// TIA Portal V20 export
FUNCTION "CallManualOperationLines_Unit1" : Void   // FC83, LAD
// stored: SetENOAutomatically false
   VAR_TEMP
      StatusEm : Array[0..7] of Struct
         Status : Array[0..40] of Word;
      END_STRUCT;
      errorIDEm : Array[0..7] of Struct
         errorID : Array[0..40] of Word;
      END_STRUCT;
      disableUnit1 : Bool;
      TempAxisCommands : "LBC_typeAxis64PosManualCommands";
      TempAxisMonitoring : "LBC_typeAxis64PosProcessValues";
      TempSoftCam : Array[0..8] of "LER_typeSoftCamParameter";
   END_VAR
   VAR CONSTANT
      MECHANIC_NAME_ENABLE : Bool;
   END_VAR
   VAR_TEMP   // added for the SCL form of the ladder/FBD networks
      _w1 : Bool;
   END_VAR
BEGIN

REGION Network 1: Unit 1 Enable Manual Operation
   // Condition to disable manual operation lines in Unit 3
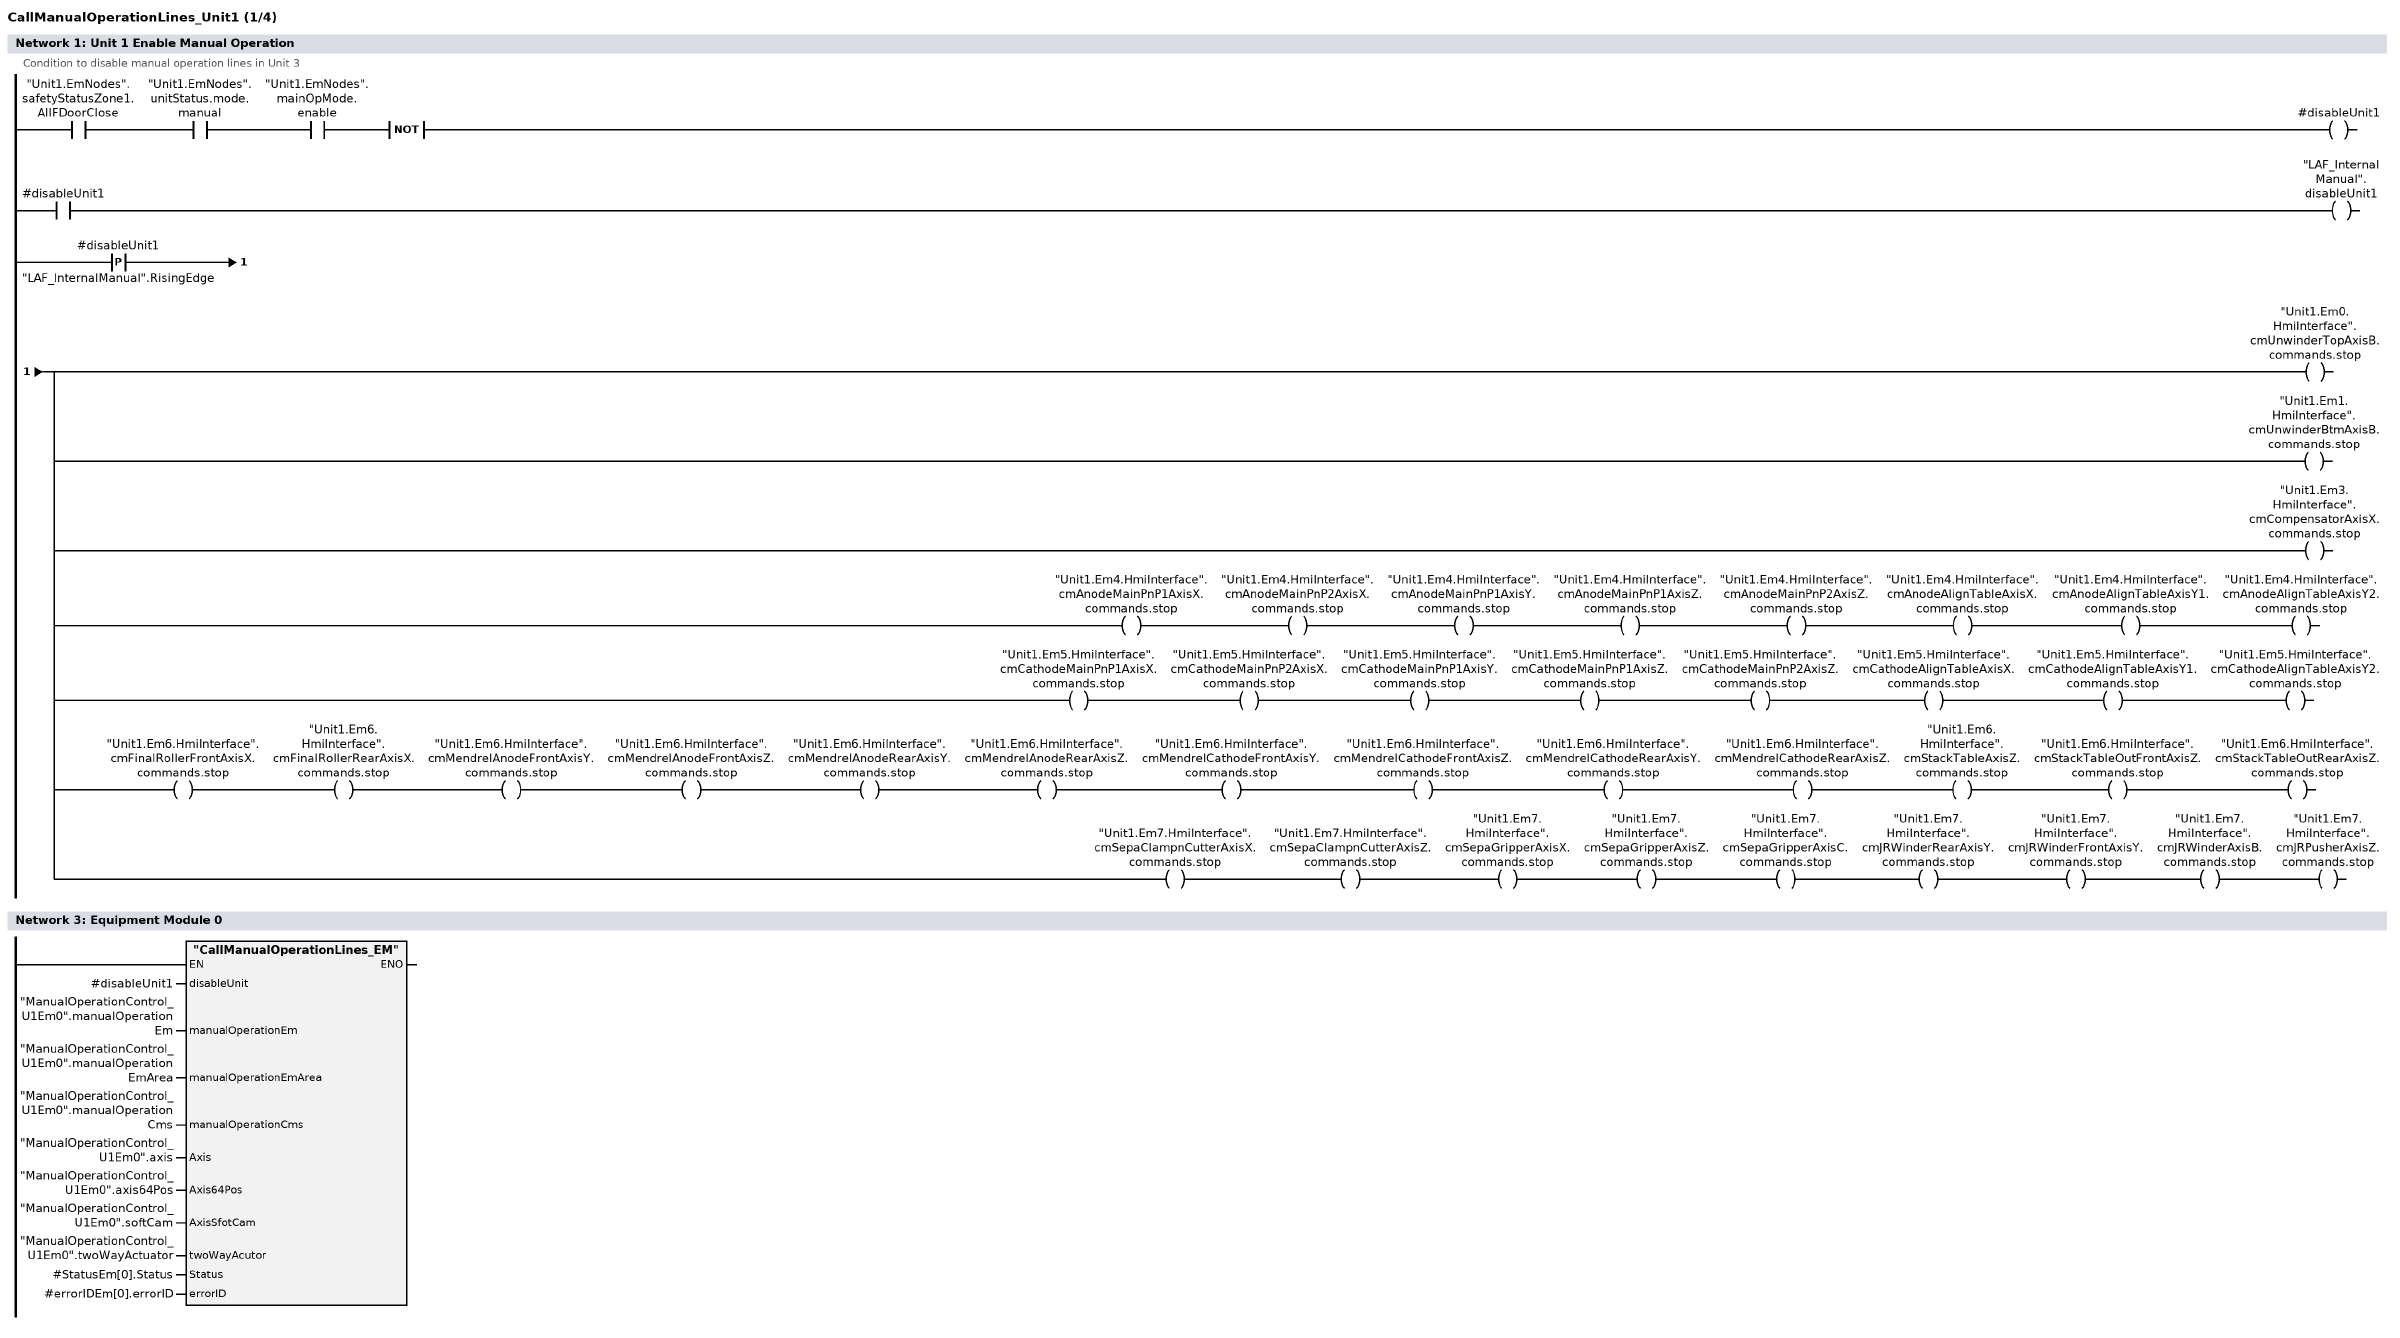
   RUNG wire#powerrail
      Contact( "Unit1.EmNodes".safetyStatusZone1.AllFDoorClose )
      Contact( "Unit1.EmNodes".unitStatus.mode.manual )
      Contact( "Unit1.EmNodes".mainOpMode.enable )
      Not()
      Coil( #disableUnit1 )
   END_RUNG
   RUNG wire#powerrail
      Contact( #disableUnit1 )
      Coil( "LAF_InternalManual".disableUnit1 )
   END_RUNG
   RUNG wire#powerrail
      P_Contact(operand := #disableUnit1, bit := "LAF_InternalManual".RisingEdge)
      wire#w1
      Coil( "Unit1.Em0.HmiInterface".cmUnwinderTopAxisB.commands.stop )
   END_RUNG
   RUNG wire#w1
      Coil( "Unit1.Em1.HmiInterface".cmUnwinderBtmAxisB.commands.stop )
   END_RUNG
   RUNG wire#w1
      Coil( "Unit1.Em3.HmiInterface".cmCompensatorAxisX.commands.stop )
   END_RUNG
   RUNG wire#w1
      Coil( "Unit1.Em4.HmiInterface".cmAnodeMainPnP1AxisX.commands.stop )
      Coil( "Unit1.Em4.HmiInterface".cmAnodeMainPnP2AxisX.commands.stop )
      Coil( "Unit1.Em4.HmiInterface".cmAnodeMainPnP1AxisY.commands.stop )
      Coil( "Unit1.Em4.HmiInterface".cmAnodeMainPnP1AxisZ.commands.stop )
      Coil( "Unit1.Em4.HmiInterface".cmAnodeMainPnP2AxisZ.commands.stop )
      Coil( "Unit1.Em4.HmiInterface".cmAnodeAlignTableAxisX.commands.stop )
      Coil( "Unit1.Em4.HmiInterface".cmAnodeAlignTableAxisY1.commands.stop )
      Coil( "Unit1.Em4.HmiInterface".cmAnodeAlignTableAxisY2.commands.stop )
   END_RUNG
   RUNG wire#w1
      Coil( "Unit1.Em5.HmiInterface".cmCathodeMainPnP1AxisX.commands.stop )
      Coil( "Unit1.Em5.HmiInterface".cmCathodeMainPnP2AxisX.commands.stop )
      Coil( "Unit1.Em5.HmiInterface".cmCathodeMainPnP1AxisY.commands.stop )
      Coil( "Unit1.Em5.HmiInterface".cmCathodeMainPnP1AxisZ.commands.stop )
      Coil( "Unit1.Em5.HmiInterface".cmCathodeMainPnP2AxisZ.commands.stop )
      Coil( "Unit1.Em5.HmiInterface".cmCathodeAlignTableAxisX.commands.stop )
      Coil( "Unit1.Em5.HmiInterface".cmCathodeAlignTableAxisY1.commands.stop )
      Coil( "Unit1.Em5.HmiInterface".cmCathodeAlignTableAxisY2.commands.stop )
   END_RUNG
   RUNG wire#w1
      Coil( "Unit1.Em6.HmiInterface".cmFinalRollerFrontAxisX.commands.stop )
      Coil( "Unit1.Em6.HmiInterface".cmFinalRollerRearAxisX.commands.stop )
      Coil( "Unit1.Em6.HmiInterface".cmMendrelAnodeFrontAxisY.commands.stop )
      Coil( "Unit1.Em6.HmiInterface".cmMendrelAnodeFrontAxisZ.commands.stop )
      Coil( "Unit1.Em6.HmiInterface".cmMendrelAnodeRearAxisY.commands.stop )
      Coil( "Unit1.Em6.HmiInterface".cmMendrelAnodeRearAxisZ.commands.stop )
      Coil( "Unit1.Em6.HmiInterface".cmMendrelCathodeFrontAxisY.commands.stop )
      Coil( "Unit1.Em6.HmiInterface".cmMendrelCathodeFrontAxisZ.commands.stop )
      Coil( "Unit1.Em6.HmiInterface".cmMendrelCathodeRearAxisY.commands.stop )
      Coil( "Unit1.Em6.HmiInterface".cmMendrelCathodeRearAxisZ.commands.stop )
      Coil( "Unit1.Em6.HmiInterface".cmStackTableAxisZ.commands.stop )
      Coil( "Unit1.Em6.HmiInterface".cmStackTableOutFrontAxisZ.commands.stop )
      Coil( "Unit1.Em6.HmiInterface".cmStackTableOutRearAxisZ.commands.stop )
   END_RUNG
   RUNG wire#w1
      Coil( "Unit1.Em7.HmiInterface".cmSepaClampnCutterAxisX.commands.stop )
      Coil( "Unit1.Em7.HmiInterface".cmSepaClampnCutterAxisZ.commands.stop )
      Coil( "Unit1.Em7.HmiInterface".cmSepaGripperAxisX.commands.stop )
      Coil( "Unit1.Em7.HmiInterface".cmSepaGripperAxisZ.commands.stop )
      Coil( "Unit1.Em7.HmiInterface".cmSepaGripperAxisC.commands.stop )
      Coil( "Unit1.Em7.HmiInterface".cmJRWinderRearAxisY.commands.stop )
      Coil( "Unit1.Em7.HmiInterface".cmJRWinderFrontAxisY.commands.stop )
      Coil( "Unit1.Em7.HmiInterface".cmJRWinderAxisB.commands.stop )
      Coil( "Unit1.Em7.HmiInterface".cmJRPusherAxisZ.commands.stop )
   END_RUNG
   // the same network as SCL:
   #disableUnit1 := NOT ("Unit1.EmNodes".safetyStatusZone1.AllFDoorClose AND "Unit1.EmNodes".unitStatus.mode.manual AND "Unit1.EmNodes".mainOpMode.enable);
   "LAF_InternalManual".disableUnit1 := #disableUnit1;
   #_w1 := #disableUnit1 AND NOT "LAF_InternalManual".RisingEdge;   // rising edge of #disableUnit1
   "LAF_InternalManual".RisingEdge := #disableUnit1;
   "Unit1.Em0.HmiInterface".cmUnwinderTopAxisB.commands.stop := #_w1;
   "Unit1.Em1.HmiInterface".cmUnwinderBtmAxisB.commands.stop := #_w1;
   "Unit1.Em3.HmiInterface".cmCompensatorAxisX.commands.stop := #_w1;
   "Unit1.Em4.HmiInterface".cmAnodeMainPnP1AxisX.commands.stop := #_w1;
   "Unit1.Em4.HmiInterface".cmAnodeMainPnP2AxisX.commands.stop := #_w1;
   "Unit1.Em4.HmiInterface".cmAnodeMainPnP1AxisY.commands.stop := #_w1;
   "Unit1.Em4.HmiInterface".cmAnodeMainPnP1AxisZ.commands.stop := #_w1;
   "Unit1.Em4.HmiInterface".cmAnodeMainPnP2AxisZ.commands.stop := #_w1;
   "Unit1.Em4.HmiInterface".cmAnodeAlignTableAxisX.commands.stop := #_w1;
   "Unit1.Em4.HmiInterface".cmAnodeAlignTableAxisY1.commands.stop := #_w1;
   "Unit1.Em4.HmiInterface".cmAnodeAlignTableAxisY2.commands.stop := #_w1;
   "Unit1.Em5.HmiInterface".cmCathodeMainPnP1AxisX.commands.stop := #_w1;
   "Unit1.Em5.HmiInterface".cmCathodeMainPnP2AxisX.commands.stop := #_w1;
   "Unit1.Em5.HmiInterface".cmCathodeMainPnP1AxisY.commands.stop := #_w1;
   "Unit1.Em5.HmiInterface".cmCathodeMainPnP1AxisZ.commands.stop := #_w1;
   "Unit1.Em5.HmiInterface".cmCathodeMainPnP2AxisZ.commands.stop := #_w1;
   "Unit1.Em5.HmiInterface".cmCathodeAlignTableAxisX.commands.stop := #_w1;
   "Unit1.Em5.HmiInterface".cmCathodeAlignTableAxisY1.commands.stop := #_w1;
   "Unit1.Em5.HmiInterface".cmCathodeAlignTableAxisY2.commands.stop := #_w1;
   "Unit1.Em6.HmiInterface".cmFinalRollerFrontAxisX.commands.stop := #_w1;
   "Unit1.Em6.HmiInterface".cmFinalRollerRearAxisX.commands.stop := #_w1;
   "Unit1.Em6.HmiInterface".cmMendrelAnodeFrontAxisY.commands.stop := #_w1;
   "Unit1.Em6.HmiInterface".cmMendrelAnodeFrontAxisZ.commands.stop := #_w1;
   "Unit1.Em6.HmiInterface".cmMendrelAnodeRearAxisY.commands.stop := #_w1;
   "Unit1.Em6.HmiInterface".cmMendrelAnodeRearAxisZ.commands.stop := #_w1;
   "Unit1.Em6.HmiInterface".cmMendrelCathodeFrontAxisY.commands.stop := #_w1;
   "Unit1.Em6.HmiInterface".cmMendrelCathodeFrontAxisZ.commands.stop := #_w1;
   "Unit1.Em6.HmiInterface".cmMendrelCathodeRearAxisY.commands.stop := #_w1;
   "Unit1.Em6.HmiInterface".cmMendrelCathodeRearAxisZ.commands.stop := #_w1;
   "Unit1.Em6.HmiInterface".cmStackTableAxisZ.commands.stop := #_w1;
   "Unit1.Em6.HmiInterface".cmStackTableOutFrontAxisZ.commands.stop := #_w1;
   "Unit1.Em6.HmiInterface".cmStackTableOutRearAxisZ.commands.stop := #_w1;
   "Unit1.Em7.HmiInterface".cmSepaClampnCutterAxisX.commands.stop := #_w1;
   "Unit1.Em7.HmiInterface".cmSepaClampnCutterAxisZ.commands.stop := #_w1;
   "Unit1.Em7.HmiInterface".cmSepaGripperAxisX.commands.stop := #_w1;
   "Unit1.Em7.HmiInterface".cmSepaGripperAxisZ.commands.stop := #_w1;
   "Unit1.Em7.HmiInterface".cmSepaGripperAxisC.commands.stop := #_w1;
   "Unit1.Em7.HmiInterface".cmJRWinderRearAxisY.commands.stop := #_w1;
   "Unit1.Em7.HmiInterface".cmJRWinderFrontAxisY.commands.stop := #_w1;
   "Unit1.Em7.HmiInterface".cmJRWinderAxisB.commands.stop := #_w1;
   "Unit1.Em7.HmiInterface".cmJRPusherAxisZ.commands.stop := #_w1;
END_REGION

REGION Network 2 (SCL): Equipment Module 0 Cms Mapping
   REGION Input Mapping
       // Axis
       "ManualOperationControl_U1Em0".axis64Pos[6].monitoring := "Unit1.Em0.HmiInterface".cmUnwinderTopAxisB.monitoring;

       "ManualOperationControl_U1Em0".axis64Pos[6].configuration := "Unit1.Em0.HmiInterface".cmUnwinderTopAxisB.configuration;
       // SoftCam
       "ManualOperationControl_U1Em0".softCam[6] := "Unit1.Em0.HmiInterface".cm.softCam.unwinderTopAxisB;

       // TwoWayActuator
       "ManualOperationControl_U1Em0".twoWayActuator[1].monitoring := "Unit1.Em0.HmiInterface".cmAirShaftTopOnOff.monitoring;
   END_REGION


   REGION Output Mapping
       // Axis
       "CallManualOperationLines_ServoPos64Commands"(ManualOperationControl := "ManualOperationControl_U1Em0".axis64Pos[6].commands,
                                                     HmiInterface => "Unit1.Em0.HmiInterface".cmUnwinderTopAxisB.commands);

       // TwoWayActuator
       "Unit1.Em0.HmiInterface".cmAirShaftTopOnOff.commands := "ManualOperationControl_U1Em0".twoWayActuator[1].commands;
   END_REGION
END_REGION

REGION Network 3: Equipment Module 0
   RUNG wire#powerrail
      "CallManualOperationLines_EM"(disableUnit := #disableUnit1, manualOperationEm := "ManualOperationControl_U1Em0".manualOperationEm, manualOperationEmArea := "ManualOperationControl_U1Em0".manualOperationEmArea, manualOperationCms := "ManualOperationControl_U1Em0".manualOperationCms, Axis := "ManualOperationControl_U1Em0".axis, Axis64Pos := "ManualOperationControl_U1Em0".axis64Pos, AxisSfotCam := "ManualOperationControl_U1Em0".softCam, twoWayAcutor := "ManualOperationControl_U1Em0".twoWayActuator, Status := #StatusEm[0].Status, errorID := #errorIDEm[0].errorID)
   END_RUNG
   // the same network as SCL:
   "CallManualOperationLines_EM"(disableUnit := #disableUnit1,
                           manualOperationEm := "ManualOperationControl_U1Em0".manualOperationEm,
                           manualOperationEmArea := "ManualOperationControl_U1Em0".manualOperationEmArea,
                           manualOperationCms := "ManualOperationControl_U1Em0".manualOperationCms,
                           Axis := "ManualOperationControl_U1Em0".axis,
                           Axis64Pos := "ManualOperationControl_U1Em0".axis64Pos,
                           AxisSfotCam := "ManualOperationControl_U1Em0".softCam,
                           twoWayAcutor := "ManualOperationControl_U1Em0".twoWayActuator,
                           Status := #StatusEm[0].Status,
                           errorID := #errorIDEm[0].errorID);
END_REGION

REGION Network 4 (SCL): Equipment Module 1 Cms Mapping
   REGION Input Mapping
       // Axis
       "ManualOperationControl_U1Em1".axis64Pos[6].monitoring := "Unit1.Em1.HmiInterface".cmUnwinderBtmAxisB.monitoring;

       "ManualOperationControl_U1Em1".axis64Pos[6].configuration := "Unit1.Em1.HmiInterface".cmUnwinderBtmAxisB.configuration;
       // SoftCam
       "ManualOperationControl_U1Em1".softCam[6] := "Unit1.Em1.HmiInterface".cm.softCam.unwinderBtmAxisB;

       // TwoWayActuator
       "ManualOperationControl_U1Em1".twoWayActuator[1].monitoring := "Unit1.Em1.HmiInterface".cmAirShaftBtmOnOff.monitoring;
   END_REGION


   REGION Output Mapping
       // Axis
       "CallManualOperationLines_ServoPos64Commands"(ManualOperationControl := "ManualOperationControl_U1Em1".axis64Pos[6].commands,
                                                     HmiInterface => "Unit1.Em1.HmiInterface".cmUnwinderBtmAxisB.commands);

       // TwoWayActuator
       "Unit1.Em0.HmiInterface".cmAirShaftTopOnOff.commands := "ManualOperationControl_U1Em0".twoWayActuator[1].commands;
   END_REGION
END_REGION

REGION Network 5: Equipment Module 1
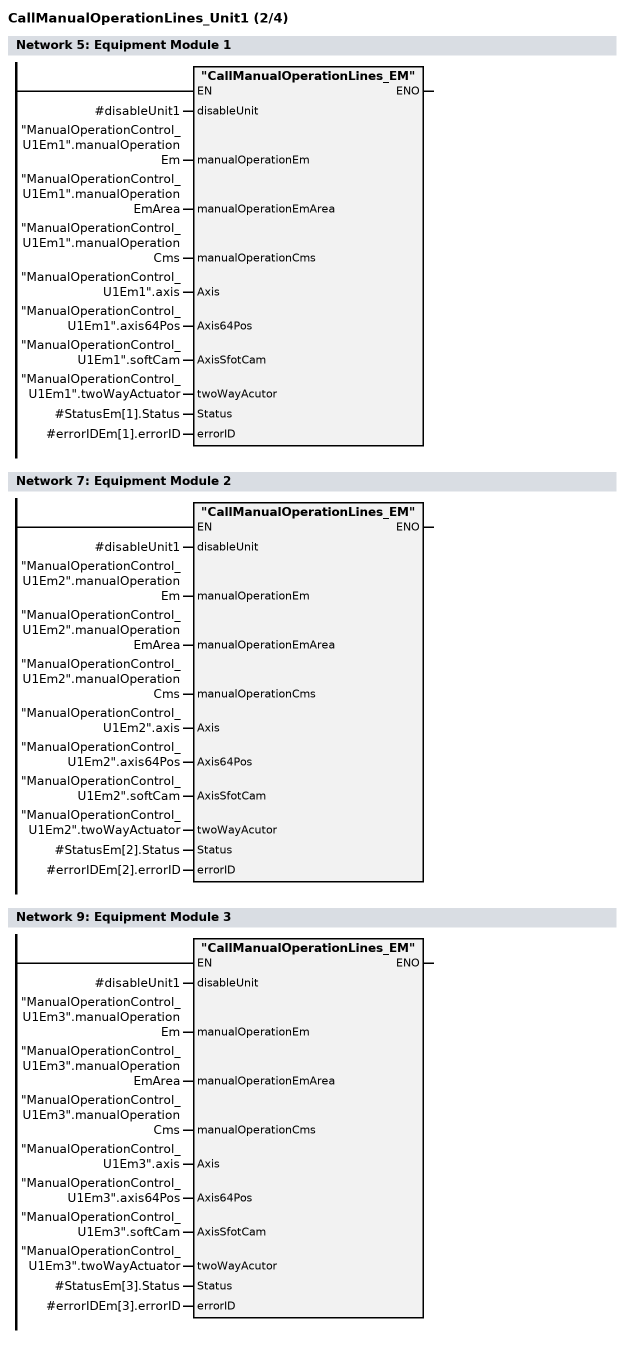
   RUNG wire#powerrail
      "CallManualOperationLines_EM"(disableUnit := #disableUnit1, manualOperationEm := "ManualOperationControl_U1Em1".manualOperationEm, manualOperationEmArea := "ManualOperationControl_U1Em1".manualOperationEmArea, manualOperationCms := "ManualOperationControl_U1Em1".manualOperationCms, Axis := "ManualOperationControl_U1Em1".axis, Axis64Pos := "ManualOperationControl_U1Em1".axis64Pos, AxisSfotCam := "ManualOperationControl_U1Em1".softCam, twoWayAcutor := "ManualOperationControl_U1Em1".twoWayActuator, Status := #StatusEm[1].Status, errorID := #errorIDEm[1].errorID)
   END_RUNG
   // the same network as SCL:
   "CallManualOperationLines_EM"(disableUnit := #disableUnit1,
                           manualOperationEm := "ManualOperationControl_U1Em1".manualOperationEm,
                           manualOperationEmArea := "ManualOperationControl_U1Em1".manualOperationEmArea,
                           manualOperationCms := "ManualOperationControl_U1Em1".manualOperationCms,
                           Axis := "ManualOperationControl_U1Em1".axis,
                           Axis64Pos := "ManualOperationControl_U1Em1".axis64Pos,
                           AxisSfotCam := "ManualOperationControl_U1Em1".softCam,
                           twoWayAcutor := "ManualOperationControl_U1Em1".twoWayActuator,
                           Status := #StatusEm[1].Status,
                           errorID := #errorIDEm[1].errorID);
END_REGION

REGION Network 6 (SCL): Equipment Module 2 Cms Mapping
   REGION Input Mapping  
       // TwoWayActuator
       "ManualOperationControl_U1Em2".twoWayActuator[1].monitoring := "Unit1.Em2.HmiInterface".cmSuctionPadTopUpDown.monitoring;
       "ManualOperationControl_U1Em2".twoWayActuator[2].monitoring := "Unit1.Em2.HmiInterface".cmSuctionPadBtmUpDown.monitoring;
       "ManualOperationControl_U1Em2".twoWayActuator[3].monitoring := "Unit1.Em2.HmiInterface".cmCutterUpDown.monitoring;
       "ManualOperationControl_U1Em2".twoWayActuator[4].monitoring := "Unit1.Em2.HmiInterface".cmTapeTopUpDown.monitoring;
       "ManualOperationControl_U1Em2".twoWayActuator[5].monitoring := "Unit1.Em2.HmiInterface".cmTapeBtmUpDown.monitoring;
       "ManualOperationControl_U1Em2".twoWayActuator[6].monitoring := "Unit1.Em2.HmiInterface".cmSpliceHeadRotateTopFwdBwd.monitoring;
       "ManualOperationControl_U1Em2".twoWayActuator[7].monitoring := "Unit1.Em2.HmiInterface".cmSpliceHeadRotateBtmFwdBwd.monitoring;
       "ManualOperationControl_U1Em2".twoWayActuator[8].monitoring := "Unit1.Em2.HmiInterface".cmSuctionPadTopLeftVaccum.monitoring;
       "ManualOperationControl_U1Em2".twoWayActuator[9].monitoring := "Unit1.Em2.HmiInterface".cmSuctionPadTopRightVaccum.monitoring;
       "ManualOperationControl_U1Em2".twoWayActuator[10].monitoring := "Unit1.Em2.HmiInterface".cmSuctionPadBtmLeftVaccum.monitoring;
       "ManualOperationControl_U1Em2".twoWayActuator[11].monitoring := "Unit1.Em2.HmiInterface".cmSuctionPadBtmRightVaccum.monitoring;
       "ManualOperationControl_U1Em2".twoWayActuator[12].monitoring := "Unit1.Em2.HmiInterface".cmSuctionPadTopTapeVaccum.monitoring;
       "ManualOperationControl_U1Em2".twoWayActuator[13].monitoring := "Unit1.Em2.HmiInterface".cmSuctionPadBtmTapeVaccum.monitoring;

   END_REGION

   REGION Output Mapping
       // TwoWayActuator
       "Unit1.Em2.HmiInterface".cmSuctionPadTopUpDown.commands := "ManualOperationControl_U1Em2".twoWayActuator[1].commands;
       "Unit1.Em2.HmiInterface".cmSuctionPadBtmUpDown.commands := "ManualOperationControl_U1Em2".twoWayActuator[2].commands;
       "Unit1.Em2.HmiInterface".cmCutterUpDown.commands := "ManualOperationControl_U1Em2".twoWayActuator[3].commands;
       "Unit1.Em2.HmiInterface".cmTapeTopUpDown.commands := "ManualOperationControl_U1Em2".twoWayActuator[4].commands;
       "Unit1.Em2.HmiInterface".cmTapeBtmUpDown.commands := "ManualOperationControl_U1Em2".twoWayActuator[5].commands;
       "Unit1.Em2.HmiInterface".cmSpliceHeadRotateTopFwdBwd.commands := "ManualOperationControl_U1Em2".twoWayActuator[6].commands;
       "Unit1.Em2.HmiInterface".cmSpliceHeadRotateBtmFwdBwd.commands := "ManualOperationControl_U1Em2".twoWayActuator[7].commands;
       "Unit1.Em2.HmiInterface".cmSuctionPadTopLeftVaccum.commands := "ManualOperationControl_U1Em2".twoWayActuator[8].commands;
       "Unit1.Em2.HmiInterface".cmSuctionPadTopRightVaccum.commands := "ManualOperationControl_U1Em2".twoWayActuator[9].commands;
       "Unit1.Em2.HmiInterface".cmSuctionPadBtmLeftVaccum.commands := "ManualOperationControl_U1Em2".twoWayActuator[10].commands;
       "Unit1.Em2.HmiInterface".cmSuctionPadBtmRightVaccum.commands := "ManualOperationControl_U1Em2".twoWayActuator[11].commands;
       "Unit1.Em2.HmiInterface".cmSuctionPadTopTapeVaccum.commands := "ManualOperationControl_U1Em2".twoWayActuator[12].commands;
       "Unit1.Em2.HmiInterface".cmSuctionPadBtmTapeVaccum.commands := "ManualOperationControl_U1Em2".twoWayActuator[13].commands;

   END_REGION
END_REGION

REGION Network 7: Equipment Module 2
   RUNG wire#powerrail
      "CallManualOperationLines_EM"(disableUnit := #disableUnit1, manualOperationEm := "ManualOperationControl_U1Em2".manualOperationEm, manualOperationEmArea := "ManualOperationControl_U1Em2".manualOperationEmArea, manualOperationCms := "ManualOperationControl_U1Em2".manualOperationCms, Axis := "ManualOperationControl_U1Em2".axis, Axis64Pos := "ManualOperationControl_U1Em2".axis64Pos, AxisSfotCam := "ManualOperationControl_U1Em2".softCam, twoWayAcutor := "ManualOperationControl_U1Em2".twoWayActuator, Status := #StatusEm[2].Status, errorID := #errorIDEm[2].errorID)
   END_RUNG
   // the same network as SCL:
   "CallManualOperationLines_EM"(disableUnit := #disableUnit1,
                           manualOperationEm := "ManualOperationControl_U1Em2".manualOperationEm,
                           manualOperationEmArea := "ManualOperationControl_U1Em2".manualOperationEmArea,
                           manualOperationCms := "ManualOperationControl_U1Em2".manualOperationCms,
                           Axis := "ManualOperationControl_U1Em2".axis,
                           Axis64Pos := "ManualOperationControl_U1Em2".axis64Pos,
                           AxisSfotCam := "ManualOperationControl_U1Em2".softCam,
                           twoWayAcutor := "ManualOperationControl_U1Em2".twoWayActuator,
                           Status := #StatusEm[2].Status,
                           errorID := #errorIDEm[2].errorID);
END_REGION

REGION Network 8 (SCL): Equipment Module 3 Cms Mapping
   REGION Input Mapping
       // Axis
       "ManualOperationControl_U1Em3".axis64Pos[6].monitoring := "Unit1.Em3.HmiInterface".cmCompensatorAxisX.monitoring;
       //"ManualOperationControl_U1Em3".axis[2].monitoring := Unit1.Em3.HmiInterface.cmSepaFeedingRollerAxisB.monitoring;
       "ManualOperationControl_U1Em3".axis64Pos[6].configuration := "Unit1.Em3.HmiInterface".cmCompensatorAxisX.configuration;
       // SoftCam
       "ManualOperationControl_U1Em3".softCam[6] := "Unit1.Em3.HmiInterface".cm.softCam.compensatorAxisX;

       // TwoWayActuator
       "ManualOperationControl_U1Em3".twoWayActuator[1].monitoring := "Unit1.Em3.HmiInterface".cmDancerFwdBwd.monitoring;
       "ManualOperationControl_U1Em3".twoWayActuator[2].monitoring := "Unit1.Em3.HmiInterface".cmSepaUnwinderIonizerTop.monitoring;
       "ManualOperationControl_U1Em3".twoWayActuator[3].monitoring := "Unit1.Em3.HmiInterface".cmSepaUnwinderIonizerBottom.monitoring;

   END_REGION

   REGION Output Mapping
       // Axis
       "CallManualOperationLines_ServoPos64Commands"(ManualOperationControl := "ManualOperationControl_U1Em3".axis64Pos[6].commands,
                                                     HmiInterface => "Unit1.Em3.HmiInterface".cmCompensatorAxisX.commands);

       // TwoWayActuator
       "Unit1.Em3.HmiInterface".cmDancerFwdBwd.commands := "ManualOperationControl_U1Em3".twoWayActuator[1].commands;
       "Unit1.Em3.HmiInterface".cmSepaUnwinderIonizerTop.commands := "ManualOperationControl_U1Em3".twoWayActuator[2].commands;
       "Unit1.Em3.HmiInterface".cmSepaUnwinderIonizerBottom.commands := "ManualOperationControl_U1Em3".twoWayActuator[3].commands;

   END_REGION
END_REGION

REGION Network 9: Equipment Module 3
   RUNG wire#powerrail
      "CallManualOperationLines_EM"(disableUnit := #disableUnit1, manualOperationEm := "ManualOperationControl_U1Em3".manualOperationEm, manualOperationEmArea := "ManualOperationControl_U1Em3".manualOperationEmArea, manualOperationCms := "ManualOperationControl_U1Em3".manualOperationCms, Axis := "ManualOperationControl_U1Em3".axis, Axis64Pos := "ManualOperationControl_U1Em3".axis64Pos, AxisSfotCam := "ManualOperationControl_U1Em3".softCam, twoWayAcutor := "ManualOperationControl_U1Em3".twoWayActuator, Status := #StatusEm[3].Status, errorID := #errorIDEm[3].errorID)
   END_RUNG
   // the same network as SCL:
   "CallManualOperationLines_EM"(disableUnit := #disableUnit1,
                           manualOperationEm := "ManualOperationControl_U1Em3".manualOperationEm,
                           manualOperationEmArea := "ManualOperationControl_U1Em3".manualOperationEmArea,
                           manualOperationCms := "ManualOperationControl_U1Em3".manualOperationCms,
                           Axis := "ManualOperationControl_U1Em3".axis,
                           Axis64Pos := "ManualOperationControl_U1Em3".axis64Pos,
                           AxisSfotCam := "ManualOperationControl_U1Em3".softCam,
                           twoWayAcutor := "ManualOperationControl_U1Em3".twoWayActuator,
                           Status := #StatusEm[3].Status,
                           errorID := #errorIDEm[3].errorID);
END_REGION

REGION Network 10 (SCL): Equipment Module 4 Cms Mapping
   REGION Input Mapping
       // Axis
       "ManualOperationControl_U1Em4".axis64Pos[6].monitoring := "Unit1.Em4.HmiInterface".cmAnodeMainPnP1AxisX.monitoring;
       "ManualOperationControl_U1Em4".axis64Pos[7].monitoring := "Unit1.Em4.HmiInterface".cmAnodeMainPnP2AxisX.monitoring;
       "ManualOperationControl_U1Em4".axis64Pos[8].monitoring := "Unit1.Em4.HmiInterface".cmAnodeMainPnP1AxisY.monitoring;
       "ManualOperationControl_U1Em4".axis64Pos[9].monitoring := "Unit1.Em4.HmiInterface".cmAnodeMainPnP1AxisZ.monitoring;
       "ManualOperationControl_U1Em4".axis64Pos[10].monitoring := "Unit1.Em4.HmiInterface".cmAnodeMainPnP2AxisZ.monitoring;
       "ManualOperationControl_U1Em4".axis64Pos[11].monitoring := "Unit1.Em4.HmiInterface".cmAnodeAlignTableAxisX.monitoring;
       "ManualOperationControl_U1Em4".axis64Pos[12].monitoring := "Unit1.Em4.HmiInterface".cmAnodeAlignTableAxisY1.monitoring;
       "ManualOperationControl_U1Em4".axis64Pos[13].monitoring := "Unit1.Em4.HmiInterface".cmAnodeAlignTableAxisY2.monitoring;

       "ManualOperationControl_U1Em4".axis64Pos[6].configuration := "Unit1.Em4.HmiInterface".cmAnodeMainPnP1AxisX.configuration;
       "ManualOperationControl_U1Em4".axis64Pos[7].configuration := "Unit1.Em4.HmiInterface".cmAnodeMainPnP2AxisX.configuration;
       "ManualOperationControl_U1Em4".axis64Pos[8].configuration := "Unit1.Em4.HmiInterface".cmAnodeMainPnP1AxisY.configuration;
       "ManualOperationControl_U1Em4".axis64Pos[9].configuration := "Unit1.Em4.HmiInterface".cmAnodeMainPnP1AxisZ.configuration;
       "ManualOperationControl_U1Em4".axis64Pos[10].configuration := "Unit1.Em4.HmiInterface".cmAnodeMainPnP2AxisZ.configuration;
       "ManualOperationControl_U1Em4".axis64Pos[11].configuration := "Unit1.Em4.HmiInterface".cmAnodeAlignTableAxisX.configuration;
       "ManualOperationControl_U1Em4".axis64Pos[12].configuration := "Unit1.Em4.HmiInterface".cmAnodeAlignTableAxisY1.configuration;
       "ManualOperationControl_U1Em4".axis64Pos[13].configuration := "Unit1.Em4.HmiInterface".cmAnodeAlignTableAxisY2.configuration;

       // SoftCam
       "ManualOperationControl_U1Em4".softCam[6] := "Unit1.Em4.HmiInterface".cm.softCam.anodeMainPnP1AxisX;
       "ManualOperationControl_U1Em4".softCam[7] := "Unit1.Em4.HmiInterface".cm.softCam.anodeMainPnP2AxisX;
       "ManualOperationControl_U1Em4".softCam[8] := "Unit1.Em4.HmiInterface".cm.softCam.anodeMainPnP1AxisY;
       "ManualOperationControl_U1Em4".softCam[9] := "Unit1.Em4.HmiInterface".cm.softCam.anodeMainPnP1AxisZ;
       "ManualOperationControl_U1Em4".softCam[10] := "Unit1.Em4.HmiInterface".cm.softCam.anodeMainPnP2AxisZ;
       "ManualOperationControl_U1Em4".softCam[11] := "Unit1.Em4.HmiInterface".cm.softCam.anodeAlignTableAxisX;
       "ManualOperationControl_U1Em4".softCam[12] := "Unit1.Em4.HmiInterface".cm.softCam.anodeAlignTableAxisY1;
       "ManualOperationControl_U1Em4".softCam[13] := "Unit1.Em4.HmiInterface".cm.softCam.anodeAlignTableAxisY2;

       // TwoWayActuator
       "ManualOperationControl_U1Em4".twoWayActuator[1].monitoring := "Unit1.Em4.HmiInterface".cmAnodeMainPnP1RotaryCwCcw.monitoring;
       "ManualOperationControl_U1Em4".twoWayActuator[2].monitoring := "Unit1.Em4.HmiInterface".cmAnodeMainPnP1SuctionPlateVacuum.monitoring;
       "ManualOperationControl_U1Em4".twoWayActuator[3].monitoring := "Unit1.Em4.HmiInterface".cmAnodeMainPnP2SuctionPlateVacuum.monitoring;
       "ManualOperationControl_U1Em4".twoWayActuator[4].monitoring := "Unit1.Em4.HmiInterface".cmAnodeAlignTableSuctionPlateVacuum.monitoring;
       "ManualOperationControl_U1Em4".twoWayActuator[5].monitoring := "Unit1.Em4.HmiInterface".cmAnodeGlassCleaning.monitoring;
       "ManualOperationControl_U1Em4".twoWayActuator[6].monitoring := "Unit1.Em4.HmiInterface".cmAnodeNgPnpUpDown.monitoring;
       "ManualOperationControl_U1Em4".twoWayActuator[7].monitoring := "Unit1.Em4.HmiInterface".cmAnodeNgPnp1stFwdBwd.monitoring;
       "ManualOperationControl_U1Em4".twoWayActuator[8].monitoring := "Unit1.Em4.HmiInterface".cmAnodeNgPnp2ndFwdBwd.monitoring;
       "ManualOperationControl_U1Em4".twoWayActuator[9].monitoring := "Unit1.Em4.HmiInterface".cmAnodeMaintenanceMovingFixFrontRearFwdBwd.monitoring;
       "ManualOperationControl_U1Em4".twoWayActuator[10].monitoring := "Unit1.Em4.HmiInterface".cmAnodeNgBoxLiftUpDown.monitoring;
       "ManualOperationControl_U1Em4".twoWayActuator[11].monitoring := "Unit1.Em4.HmiInterface".cmAnodeNgBoxLockUpDown.monitoring;
       "ManualOperationControl_U1Em4".twoWayActuator[12].monitoring := "Unit1.Em4.HmiInterface".cmAnodeNgPnpVaccum.monitoring;
       "ManualOperationControl_U1Em4".twoWayActuator[13].monitoring := "Unit1.Em4.HmiInterface".cmAnodeConveyorCoverFwdBwd.monitoring;

   END_REGION


   REGION Output Mapping
       // Axis

       "CallManualOperationLines_ServoPos64Commands"(ManualOperationControl := "ManualOperationControl_U1Em4".axis64Pos[6].commands,
                                                     HmiInterface => "Unit1.Em4.HmiInterface".cmAnodeMainPnP1AxisX.commands);

       "CallManualOperationLines_ServoPos64Commands"(ManualOperationControl := "ManualOperationControl_U1Em4".axis64Pos[7].commands,
                                                     HmiInterface => "Unit1.Em4.HmiInterface".cmAnodeMainPnP2AxisX.commands);

       "CallManualOperationLines_ServoPos64Commands"(ManualOperationControl := "ManualOperationControl_U1Em4".axis64Pos[8].commands,
                                                     HmiInterface => "Unit1.Em4.HmiInterface".cmAnodeMainPnP1AxisY.commands);

       "CallManualOperationLines_ServoPos64Commands"(ManualOperationControl := "ManualOperationControl_U1Em4".axis64Pos[9].commands,
                                                     HmiInterface => "Unit1.Em4.HmiInterface".cmAnodeMainPnP1AxisZ.commands);

       "CallManualOperationLines_ServoPos64Commands"(ManualOperationControl := "ManualOperationControl_U1Em4".axis64Pos[10].commands,
                                                     HmiInterface => "Unit1.Em4.HmiInterface".cmAnodeMainPnP2AxisZ.commands);

       "CallManualOperationLines_ServoPos64Commands"(ManualOperationControl := "ManualOperationControl_U1Em4".axis64Pos[11].commands,
                                                     HmiInterface => "Unit1.Em4.HmiInterface".cmAnodeAlignTableAxisX.commands);

       "CallManualOperationLines_ServoPos64Commands"(ManualOperationControl := "ManualOperationControl_U1Em4".axis64Pos[12].commands,
                                                     HmiInterface => "Unit1.Em4.HmiInterface".cmAnodeAlignTableAxisY1.commands);

       "CallManualOperationLines_ServoPos64Commands"(ManualOperationControl := "ManualOperationControl_U1Em4".axis64Pos[13].commands,
                                                     HmiInterface => "Unit1.Em4.HmiInterface".cmAnodeAlignTableAxisY2.commands);

       // TwoWayActuator
       "Unit1.Em4.HmiInterface".cmAnodeMainPnP1RotaryCwCcw.commands := "ManualOperationControl_U1Em4".twoWayActuator[1].commands;
       "Unit1.Em4.HmiInterface".cmAnodeMainPnP1SuctionPlateVacuum.commands := "ManualOperationControl_U1Em4".twoWayActuator[2].commands;
       "Unit1.Em4.HmiInterface".cmAnodeMainPnP2SuctionPlateVacuum.commands := "ManualOperationControl_U1Em4".twoWayActuator[3].commands;
       "Unit1.Em4.HmiInterface".cmAnodeAlignTableSuctionPlateVacuum.commands := "ManualOperationControl_U1Em4".twoWayActuator[4].commands;
       "Unit1.Em4.HmiInterface".cmAnodeGlassCleaning.commands := "ManualOperationControl_U1Em4".twoWayActuator[5].commands;
       "Unit1.Em4.HmiInterface".cmAnodeNgPnpUpDown.commands := "ManualOperationControl_U1Em4".twoWayActuator[6].commands;
       "Unit1.Em4.HmiInterface".cmAnodeNgPnp1stFwdBwd.commands := "ManualOperationControl_U1Em4".twoWayActuator[7].commands;
       "Unit1.Em4.HmiInterface".cmAnodeNgPnp2ndFwdBwd.commands := "ManualOperationControl_U1Em4".twoWayActuator[8].commands;
       "Unit1.Em4.HmiInterface".cmAnodeMaintenanceMovingFixFrontRearFwdBwd.commands := "ManualOperationControl_U1Em4".twoWayActuator[9].commands;
       "Unit1.Em4.HmiInterface".cmAnodeNgBoxLiftUpDown.commands := "ManualOperationControl_U1Em4".twoWayActuator[10].commands;
       "Unit1.Em4.HmiInterface".cmAnodeNgBoxLockUpDown.commands := "ManualOperationControl_U1Em4".twoWayActuator[11].commands;
       "Unit1.Em4.HmiInterface".cmAnodeNgPnpVaccum.commands := "ManualOperationControl_U1Em4".twoWayActuator[12].commands;
       "Unit1.Em4.HmiInterface".cmAnodeConveyorCoverFwdBwd.commands := "ManualOperationControl_U1Em4".twoWayActuator[13].commands;

   END_REGION
END_REGION

REGION Network 11: Equipment Module 4
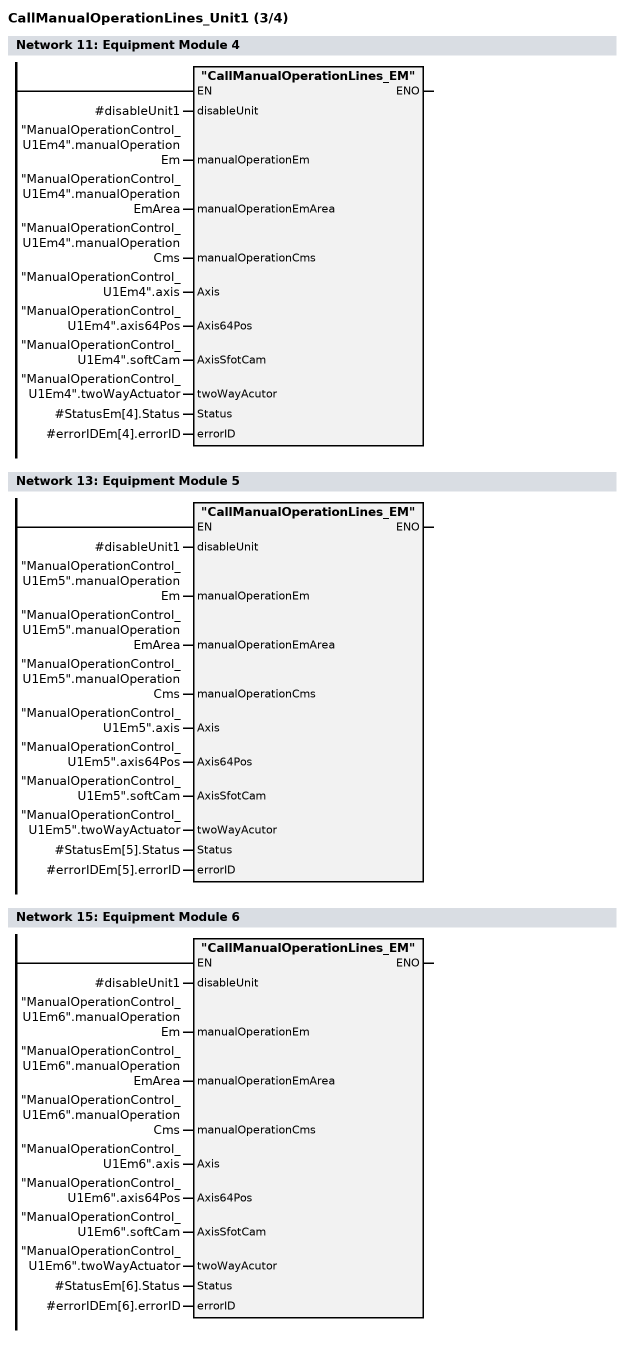
   RUNG wire#powerrail
      "CallManualOperationLines_EM"(disableUnit := #disableUnit1, manualOperationEm := "ManualOperationControl_U1Em4".manualOperationEm, manualOperationEmArea := "ManualOperationControl_U1Em4".manualOperationEmArea, manualOperationCms := "ManualOperationControl_U1Em4".manualOperationCms, Axis := "ManualOperationControl_U1Em4".axis, Axis64Pos := "ManualOperationControl_U1Em4".axis64Pos, AxisSfotCam := "ManualOperationControl_U1Em4".softCam, twoWayAcutor := "ManualOperationControl_U1Em4".twoWayActuator, Status := #StatusEm[4].Status, errorID := #errorIDEm[4].errorID)
   END_RUNG
   // the same network as SCL:
   "CallManualOperationLines_EM"(disableUnit := #disableUnit1,
                           manualOperationEm := "ManualOperationControl_U1Em4".manualOperationEm,
                           manualOperationEmArea := "ManualOperationControl_U1Em4".manualOperationEmArea,
                           manualOperationCms := "ManualOperationControl_U1Em4".manualOperationCms,
                           Axis := "ManualOperationControl_U1Em4".axis,
                           Axis64Pos := "ManualOperationControl_U1Em4".axis64Pos,
                           AxisSfotCam := "ManualOperationControl_U1Em4".softCam,
                           twoWayAcutor := "ManualOperationControl_U1Em4".twoWayActuator,
                           Status := #StatusEm[4].Status,
                           errorID := #errorIDEm[4].errorID);
END_REGION

REGION Network 12 (SCL): Equipment Module 5 Cms Mapping
   REGION Input Mapping
       // Axis
       "ManualOperationControl_U1Em5".axis64Pos[6].monitoring := "Unit1.Em5.HmiInterface".cmCathodeMainPnP1AxisX.monitoring;
       "ManualOperationControl_U1Em5".axis64Pos[7].monitoring := "Unit1.Em5.HmiInterface".cmCathodeMainPnP2AxisX.monitoring;
       "ManualOperationControl_U1Em5".axis64Pos[8].monitoring := "Unit1.Em5.HmiInterface".cmCathodeMainPnP1AxisY.monitoring;
       "ManualOperationControl_U1Em5".axis64Pos[9].monitoring := "Unit1.Em5.HmiInterface".cmCathodeMainPnP1AxisZ.monitoring;
       "ManualOperationControl_U1Em5".axis64Pos[10].monitoring := "Unit1.Em5.HmiInterface".cmCathodeMainPnP2AxisZ.monitoring;
       "ManualOperationControl_U1Em5".axis64Pos[11].monitoring := "Unit1.Em5.HmiInterface".cmCathodeAlignTableAxisX.monitoring;
       "ManualOperationControl_U1Em5".axis64Pos[12].monitoring := "Unit1.Em5.HmiInterface".cmCathodeAlignTableAxisY1.monitoring;
       "ManualOperationControl_U1Em5".axis64Pos[13].monitoring := "Unit1.Em5.HmiInterface".cmCathodeAlignTableAxisY2.monitoring;

       "ManualOperationControl_U1Em5".axis64Pos[6].configuration := "Unit1.Em5.HmiInterface".cmCathodeMainPnP1AxisX.configuration;
       "ManualOperationControl_U1Em5".axis64Pos[7].configuration := "Unit1.Em5.HmiInterface".cmCathodeMainPnP2AxisX.configuration;
       "ManualOperationControl_U1Em5".axis64Pos[8].configuration := "Unit1.Em5.HmiInterface".cmCathodeMainPnP1AxisY.configuration;
       "ManualOperationControl_U1Em5".axis64Pos[9].configuration := "Unit1.Em5.HmiInterface".cmCathodeMainPnP1AxisZ.configuration;
       "ManualOperationControl_U1Em5".axis64Pos[10].configuration := "Unit1.Em5.HmiInterface".cmCathodeMainPnP2AxisZ.configuration;
       "ManualOperationControl_U1Em5".axis64Pos[11].configuration := "Unit1.Em5.HmiInterface".cmCathodeAlignTableAxisX.configuration;
       "ManualOperationControl_U1Em5".axis64Pos[12].configuration := "Unit1.Em5.HmiInterface".cmCathodeAlignTableAxisY1.configuration;
       "ManualOperationControl_U1Em5".axis64Pos[13].configuration := "Unit1.Em5.HmiInterface".cmCathodeAlignTableAxisY2.configuration;
       // SoftCam
       "ManualOperationControl_U1Em5".softCam[6] := "Unit1.Em5.HmiInterface".cm.softCam.cathodeMainPnP1AxisX;
       "ManualOperationControl_U1Em5".softCam[7] := "Unit1.Em5.HmiInterface".cm.softCam.cathodeMainPnP2AxisX;
       "ManualOperationControl_U1Em5".softCam[8] := "Unit1.Em5.HmiInterface".cm.softCam.cathodeMainPnP1AxisY;
       "ManualOperationControl_U1Em5".softCam[9] := "Unit1.Em5.HmiInterface".cm.softCam.cathodeMainPnP1AxisZ;
       "ManualOperationControl_U1Em5".softCam[10] := "Unit1.Em5.HmiInterface".cm.softCam.cathodeMainPnP2AxisZ;
       "ManualOperationControl_U1Em5".softCam[11] := "Unit1.Em5.HmiInterface".cm.softCam.cathodeAlignTableAxisX;
       "ManualOperationControl_U1Em5".softCam[12] := "Unit1.Em5.HmiInterface".cm.softCam.cathodeAlignTableAxisY1;
       "ManualOperationControl_U1Em5".softCam[13] := "Unit1.Em5.HmiInterface".cm.softCam.cathodeAlignTableAxisY2;

       // TwoWayActuator
       "ManualOperationControl_U1Em5".twoWayActuator[1].monitoring := "Unit1.Em5.HmiInterface".cmCathodeMainPnP1RotaryCwCcw.monitoring;
       "ManualOperationControl_U1Em5".twoWayActuator[2].monitoring := "Unit1.Em5.HmiInterface".cmCathodeMainPnP1SuctionPlateVacuum.monitoring;
       "ManualOperationControl_U1Em5".twoWayActuator[3].monitoring := "Unit1.Em5.HmiInterface".cmCathodeMainPnP2SuctionPlateVacuum.monitoring;
       "ManualOperationControl_U1Em5".twoWayActuator[4].monitoring := "Unit1.Em5.HmiInterface".cmCathodeAlignTableSuctionPlateVacuum.monitoring;
       "ManualOperationControl_U1Em5".twoWayActuator[5].monitoring := "Unit1.Em5.HmiInterface".cmCathodeGlassCleaning.monitoring;
       "ManualOperationControl_U1Em5".twoWayActuator[6].monitoring := "Unit1.Em5.HmiInterface".cmCathodeNgPnpUpDown.monitoring;
       "ManualOperationControl_U1Em5".twoWayActuator[7].monitoring := "Unit1.Em5.HmiInterface".cmCathodeNgPnp1stFwdBwd.monitoring;
       "ManualOperationControl_U1Em5".twoWayActuator[8].monitoring := "Unit1.Em5.HmiInterface".cmCathodeNgPnp2ndFwdBwd.monitoring;
       "ManualOperationControl_U1Em5".twoWayActuator[9].monitoring := "Unit1.Em5.HmiInterface".cmCathodeMaintenanceMovingFixFrontRearFwdBwd.monitoring;
       "ManualOperationControl_U1Em5".twoWayActuator[10].monitoring := "Unit1.Em5.HmiInterface".cmCathodeNgBoxLiftUpDown.monitoring;
       "ManualOperationControl_U1Em5".twoWayActuator[11].monitoring := "Unit1.Em5.HmiInterface".cmCathodeNgBoxLockUpDown.monitoring;
       "ManualOperationControl_U1Em5".twoWayActuator[12].monitoring := "Unit1.Em5.HmiInterface".cmCathodeNgPnpVaccum.monitoring;
       "ManualOperationControl_U1Em5".twoWayActuator[13].monitoring := "Unit1.Em5.HmiInterface".cmCathodeConveyorCoverFwdBwd.monitoring;

   END_REGION


   REGION Output Mapping
       // Axis
       "CallManualOperationLines_ServoPos64Commands"(ManualOperationControl := "ManualOperationControl_U1Em5".axis64Pos[6].commands,
                                                     HmiInterface => "Unit1.Em5.HmiInterface".cmCathodeMainPnP1AxisX.commands);

       "CallManualOperationLines_ServoPos64Commands"(ManualOperationControl := "ManualOperationControl_U1Em5".axis64Pos[7].commands,
                                                     HmiInterface => "Unit1.Em5.HmiInterface".cmCathodeMainPnP2AxisX.commands);

       "CallManualOperationLines_ServoPos64Commands"(ManualOperationControl := "ManualOperationControl_U1Em5".axis64Pos[8].commands,
                                                     HmiInterface => "Unit1.Em5.HmiInterface".cmCathodeMainPnP1AxisY.commands);

       "CallManualOperationLines_ServoPos64Commands"(ManualOperationControl := "ManualOperationControl_U1Em5".axis64Pos[9].commands,
                                                     HmiInterface => "Unit1.Em5.HmiInterface".cmCathodeMainPnP1AxisZ.commands);

       "CallManualOperationLines_ServoPos64Commands"(ManualOperationControl := "ManualOperationControl_U1Em5".axis64Pos[10].commands,
                                                     HmiInterface => "Unit1.Em5.HmiInterface".cmCathodeMainPnP2AxisZ.commands);

       "CallManualOperationLines_ServoPos64Commands"(ManualOperationControl := "ManualOperationControl_U1Em5".axis64Pos[11].commands,
                                                     HmiInterface => "Unit1.Em5.HmiInterface".cmCathodeAlignTableAxisX.commands);

       "CallManualOperationLines_ServoPos64Commands"(ManualOperationControl := "ManualOperationControl_U1Em5".axis64Pos[12].commands,
                                                     HmiInterface => "Unit1.Em5.HmiInterface".cmCathodeAlignTableAxisY1.commands);

       "CallManualOperationLines_ServoPos64Commands"(ManualOperationControl := "ManualOperationControl_U1Em5".axis64Pos[13].commands,
                                                     HmiInterface => "Unit1.Em5.HmiInterface".cmCathodeAlignTableAxisY2.commands);

       // TwoWayActuator
       "Unit1.Em5.HmiInterface".cmCathodeMainPnP1RotaryCwCcw.commands := "ManualOperationControl_U1Em5".twoWayActuator[1].commands;
       "Unit1.Em5.HmiInterface".cmCathodeMainPnP1SuctionPlateVacuum.commands := "ManualOperationControl_U1Em5".twoWayActuator[2].commands;
       "Unit1.Em5.HmiInterface".cmCathodeMainPnP2SuctionPlateVacuum.commands := "ManualOperationControl_U1Em5".twoWayActuator[3].commands;
       "Unit1.Em5.HmiInterface".cmCathodeAlignTableSuctionPlateVacuum.commands := "ManualOperationControl_U1Em5".twoWayActuator[4].commands;
       "Unit1.Em5.HmiInterface".cmCathodeGlassCleaning.commands := "ManualOperationControl_U1Em5".twoWayActuator[5].commands;
       "Unit1.Em5.HmiInterface".cmCathodeNgPnpUpDown.commands := "ManualOperationControl_U1Em5".twoWayActuator[6].commands;
       "Unit1.Em5.HmiInterface".cmCathodeNgPnp1stFwdBwd.commands := "ManualOperationControl_U1Em5".twoWayActuator[7].commands;
       "Unit1.Em5.HmiInterface".cmCathodeNgPnp2ndFwdBwd.commands := "ManualOperationControl_U1Em5".twoWayActuator[8].commands;
       "Unit1.Em5.HmiInterface".cmCathodeMaintenanceMovingFixFrontRearFwdBwd.commands := "ManualOperationControl_U1Em5".twoWayActuator[9].commands;
       "Unit1.Em5.HmiInterface".cmCathodeNgBoxLiftUpDown.commands := "ManualOperationControl_U1Em5".twoWayActuator[10].commands;
       "Unit1.Em5.HmiInterface".cmCathodeNgBoxLockUpDown.commands := "ManualOperationControl_U1Em5".twoWayActuator[11].commands;
       "Unit1.Em5.HmiInterface".cmCathodeNgPnpVaccum.commands := "ManualOperationControl_U1Em5".twoWayActuator[12].commands;
       "Unit1.Em5.HmiInterface".cmCathodeConveyorCoverFwdBwd.commands := "ManualOperationControl_U1Em5".twoWayActuator[13].commands;

   END_REGION
END_REGION

REGION Network 13: Equipment Module 5
   RUNG wire#powerrail
      "CallManualOperationLines_EM"(disableUnit := #disableUnit1, manualOperationEm := "ManualOperationControl_U1Em5".manualOperationEm, manualOperationEmArea := "ManualOperationControl_U1Em5".manualOperationEmArea, manualOperationCms := "ManualOperationControl_U1Em5".manualOperationCms, Axis := "ManualOperationControl_U1Em5".axis, Axis64Pos := "ManualOperationControl_U1Em5".axis64Pos, AxisSfotCam := "ManualOperationControl_U1Em5".softCam, twoWayAcutor := "ManualOperationControl_U1Em5".twoWayActuator, Status := #StatusEm[5].Status, errorID := #errorIDEm[5].errorID)
   END_RUNG
   // the same network as SCL:
   "CallManualOperationLines_EM"(disableUnit := #disableUnit1,
                           manualOperationEm := "ManualOperationControl_U1Em5".manualOperationEm,
                           manualOperationEmArea := "ManualOperationControl_U1Em5".manualOperationEmArea,
                           manualOperationCms := "ManualOperationControl_U1Em5".manualOperationCms,
                           Axis := "ManualOperationControl_U1Em5".axis,
                           Axis64Pos := "ManualOperationControl_U1Em5".axis64Pos,
                           AxisSfotCam := "ManualOperationControl_U1Em5".softCam,
                           twoWayAcutor := "ManualOperationControl_U1Em5".twoWayActuator,
                           Status := #StatusEm[5].Status,
                           errorID := #errorIDEm[5].errorID);
END_REGION

REGION Network 14 (SCL): Equipment Module 6 Cms Mapping
   REGION Input Mapping
       // Axis
       "ManualOperationControl_U1Em6".axis64Pos[6].monitoring := "Unit1.Em6.HmiInterface".cmFinalRollerFrontAxisX.monitoring;
       "ManualOperationControl_U1Em6".axis64Pos[7].monitoring := "Unit1.Em6.HmiInterface".cmFinalRollerRearAxisX.monitoring;
       "ManualOperationControl_U1Em6".axis64Pos[8].monitoring := "Unit1.Em6.HmiInterface".cmMendrelCathodeFrontAxisY.monitoring;
       "ManualOperationControl_U1Em6".axis64Pos[9].monitoring := "Unit1.Em6.HmiInterface".cmMendrelCathodeFrontAxisZ.monitoring;
       "ManualOperationControl_U1Em6".axis64Pos[10].monitoring := "Unit1.Em6.HmiInterface".cmMendrelAnodeFrontAxisY.monitoring;
       "ManualOperationControl_U1Em6".axis64Pos[11].monitoring := "Unit1.Em6.HmiInterface".cmMendrelAnodeFrontAxisZ.monitoring;
       "ManualOperationControl_U1Em6".axis64Pos[12].monitoring := "Unit1.Em6.HmiInterface".cmMendrelCathodeRearAxisY.monitoring;
       "ManualOperationControl_U1Em6".axis64Pos[13].monitoring := "Unit1.Em6.HmiInterface".cmMendrelCathodeRearAxisZ.monitoring;
       "ManualOperationControl_U1Em6".axis64Pos[14].monitoring := "Unit1.Em6.HmiInterface".cmMendrelAnodeRearAxisY.monitoring;
       "ManualOperationControl_U1Em6".axis64Pos[15].monitoring := "Unit1.Em6.HmiInterface".cmMendrelAnodeRearAxisZ.monitoring;
       "ManualOperationControl_U1Em6".axis64Pos[16].monitoring := "Unit1.Em6.HmiInterface".cmStackTableAxisZ.monitoring;
       "ManualOperationControl_U1Em6".axis64Pos[17].monitoring := "Unit1.Em6.HmiInterface".cmStackTableOutFrontAxisZ.monitoring;
       "ManualOperationControl_U1Em6".axis64Pos[18].monitoring := "Unit1.Em6.HmiInterface".cmStackTableOutRearAxisZ.monitoring;

       "ManualOperationControl_U1Em6".axis64Pos[6].configuration := "Unit1.Em6.HmiInterface".cmFinalRollerFrontAxisX.configuration;
       "ManualOperationControl_U1Em6".axis64Pos[7].configuration := "Unit1.Em6.HmiInterface".cmFinalRollerRearAxisX.configuration;
       "ManualOperationControl_U1Em6".axis64Pos[8].configuration := "Unit1.Em6.HmiInterface".cmMendrelCathodeFrontAxisY.configuration;
       "ManualOperationControl_U1Em6".axis64Pos[9].configuration := "Unit1.Em6.HmiInterface".cmMendrelCathodeFrontAxisZ.configuration;
       "ManualOperationControl_U1Em6".axis64Pos[10].configuration := "Unit1.Em6.HmiInterface".cmMendrelAnodeFrontAxisY.configuration;
       "ManualOperationControl_U1Em6".axis64Pos[11].configuration := "Unit1.Em6.HmiInterface".cmMendrelAnodeFrontAxisZ.configuration;
       "ManualOperationControl_U1Em6".axis64Pos[12].configuration := "Unit1.Em6.HmiInterface".cmMendrelCathodeRearAxisY.configuration;
       "ManualOperationControl_U1Em6".axis64Pos[13].configuration := "Unit1.Em6.HmiInterface".cmMendrelCathodeRearAxisZ.configuration;
       "ManualOperationControl_U1Em6".axis64Pos[14].configuration := "Unit1.Em6.HmiInterface".cmMendrelAnodeRearAxisY.configuration;
       "ManualOperationControl_U1Em6".axis64Pos[15].configuration := "Unit1.Em6.HmiInterface".cmMendrelAnodeRearAxisZ.configuration;
       "ManualOperationControl_U1Em6".axis64Pos[16].configuration := "Unit1.Em6.HmiInterface".cmStackTableAxisZ.configuration;
       "ManualOperationControl_U1Em6".axis64Pos[17].configuration := "Unit1.Em6.HmiInterface".cmStackTableOutFrontAxisZ.configuration;
       "ManualOperationControl_U1Em6".axis64Pos[18].configuration := "Unit1.Em6.HmiInterface".cmStackTableOutRearAxisZ.configuration;

       // SoftCam
       "ManualOperationControl_U1Em6".softCam[6] := "Unit1.Em6.HmiInterface".cm.softCam.finalRollerFrontAxisX;
       "ManualOperationControl_U1Em6".softCam[7] := "Unit1.Em6.HmiInterface".cm.softCam.finalRollerRearAxisX;
       "ManualOperationControl_U1Em6".softCam[8] := "Unit1.Em6.HmiInterface".cm.softCam.mendrelAnodeFrontAxisY;
       "ManualOperationControl_U1Em6".softCam[9] := "Unit1.Em6.HmiInterface".cm.softCam.mendrelAnodeFrontAxisZ;
       "ManualOperationControl_U1Em6".softCam[10] := "Unit1.Em6.HmiInterface".cm.softCam.mendrelAnodeRearAxisY;
       "ManualOperationControl_U1Em6".softCam[11] := "Unit1.Em6.HmiInterface".cm.softCam.mendrelAnodeRearAxisZ;
       "ManualOperationControl_U1Em6".softCam[12] := "Unit1.Em6.HmiInterface".cm.softCam.mendrelCathodeFrontAxisY;
       "ManualOperationControl_U1Em6".softCam[13] := "Unit1.Em6.HmiInterface".cm.softCam.mendrelCathodeFrontAxisZ;
       "ManualOperationControl_U1Em6".softCam[14] := "Unit1.Em6.HmiInterface".cm.softCam.mendrelCathodeRearAxisY;
       "ManualOperationControl_U1Em6".softCam[15] := "Unit1.Em6.HmiInterface".cm.softCam.mendrelCathodeRearAxisZ;
       "ManualOperationControl_U1Em6".softCam[16] := "Unit1.Em6.HmiInterface".cm.softCam.stackTableAxisZ;
       "ManualOperationControl_U1Em6".softCam[17] := "Unit1.Em6.HmiInterface".cm.softCam.stackTableOutFrontAxisZ;
       "ManualOperationControl_U1Em6".softCam[18] := "Unit1.Em6.HmiInterface".cm.softCam.stackTableOutRearAxisZ;

       // TwoWayActuator
       "ManualOperationControl_U1Em6".twoWayActuator[1].monitoring := "Unit1.Em6.HmiInterface".cmMendrelCathodeFrontClamp.monitoring;
       "ManualOperationControl_U1Em6".twoWayActuator[2].monitoring := "Unit1.Em6.HmiInterface".cmMendrelAnodeFrontClamp.monitoring;
       "ManualOperationControl_U1Em6".twoWayActuator[3].monitoring := "Unit1.Em6.HmiInterface".cmMendrelCathodeRearClamp.monitoring;
       "ManualOperationControl_U1Em6".twoWayActuator[4].monitoring := "Unit1.Em6.HmiInterface".cmMendrelAnodeRearClamp.monitoring;
       "ManualOperationControl_U1Em6".twoWayActuator[5].monitoring := "Unit1.Em6.HmiInterface".cmStackTableVaccum.monitoring;
       "ManualOperationControl_U1Em6".twoWayActuator[6].monitoring := "Unit1.Em6.HmiInterface".cmStackTableGapPadUpDown.monitoring;

   END_REGION


   REGION Output Mapping
       // Axis
       "CallManualOperationLines_ServoPos64Commands"(ManualOperationControl := "ManualOperationControl_U1Em6".axis64Pos[6].commands,
                                                     HmiInterface => "Unit1.Em6.HmiInterface".cmFinalRollerFrontAxisX.commands);

       "CallManualOperationLines_ServoPos64Commands"(ManualOperationControl := "ManualOperationControl_U1Em6".axis64Pos[7].commands,
                                                     HmiInterface => "Unit1.Em6.HmiInterface".cmFinalRollerRearAxisX.commands);

       "CallManualOperationLines_ServoPos64Commands"(ManualOperationControl := "ManualOperationControl_U1Em6".axis64Pos[8].commands,
                                                     HmiInterface => "Unit1.Em6.HmiInterface".cmMendrelCathodeFrontAxisY.commands);

       "CallManualOperationLines_ServoPos64Commands"(ManualOperationControl := "ManualOperationControl_U1Em6".axis64Pos[9].commands,
                                                     HmiInterface => "Unit1.Em6.HmiInterface".cmMendrelCathodeFrontAxisZ.commands);

       "CallManualOperationLines_ServoPos64Commands"(ManualOperationControl := "ManualOperationControl_U1Em6".axis64Pos[10].commands,
                                                     HmiInterface => "Unit1.Em6.HmiInterface".cmMendrelAnodeFrontAxisY.commands);

       "CallManualOperationLines_ServoPos64Commands"(ManualOperationControl := "ManualOperationControl_U1Em6".axis64Pos[11].commands,
                                                     HmiInterface => "Unit1.Em6.HmiInterface".cmMendrelAnodeFrontAxisZ.commands);

       "CallManualOperationLines_ServoPos64Commands"(ManualOperationControl := "ManualOperationControl_U1Em6".axis64Pos[12].commands,
                                                     HmiInterface => "Unit1.Em6.HmiInterface".cmMendrelCathodeRearAxisY.commands);

       "CallManualOperationLines_ServoPos64Commands"(ManualOperationControl := "ManualOperationControl_U1Em6".axis64Pos[13].commands,
                                                     HmiInterface => "Unit1.Em6.HmiInterface".cmMendrelCathodeRearAxisZ.commands);

       "CallManualOperationLines_ServoPos64Commands"(ManualOperationControl := "ManualOperationControl_U1Em6".axis64Pos[14].commands,
                                                     HmiInterface => "Unit1.Em6.HmiInterface".cmMendrelAnodeRearAxisY.commands);

       "CallManualOperationLines_ServoPos64Commands"(ManualOperationControl := "ManualOperationControl_U1Em6".axis64Pos[15].commands,
                                                     HmiInterface => "Unit1.Em6.HmiInterface".cmMendrelAnodeRearAxisZ.commands);

       "CallManualOperationLines_ServoPos64Commands"(ManualOperationControl := "ManualOperationControl_U1Em6".axis64Pos[16].commands,
                                                     HmiInterface => "Unit1.Em6.HmiInterface".cmStackTableAxisZ.commands);

       "CallManualOperationLines_ServoPos64Commands"(ManualOperationControl := "ManualOperationControl_U1Em6".axis64Pos[17].commands,
                                                     HmiInterface => "Unit1.Em6.HmiInterface".cmStackTableOutFrontAxisZ.commands);

       "CallManualOperationLines_ServoPos64Commands"(ManualOperationControl := "ManualOperationControl_U1Em6".axis64Pos[18].commands,
                                                     HmiInterface => "Unit1.Em6.HmiInterface".cmStackTableOutRearAxisZ.commands);

       // TwoWayActuator
       "Unit1.Em6.HmiInterface".cmMendrelCathodeFrontClamp.commands := "ManualOperationControl_U1Em6".twoWayActuator[1].commands;
       "Unit1.Em6.HmiInterface".cmMendrelAnodeFrontClamp.commands := "ManualOperationControl_U1Em6".twoWayActuator[2].commands;
       "Unit1.Em6.HmiInterface".cmMendrelCathodeRearClamp.commands := "ManualOperationControl_U1Em6".twoWayActuator[3].commands;
       "Unit1.Em6.HmiInterface".cmMendrelAnodeRearClamp.commands := "ManualOperationControl_U1Em6".twoWayActuator[4].commands;
       "Unit1.Em6.HmiInterface".cmStackTableVaccum.commands := "ManualOperationControl_U1Em6".twoWayActuator[5].commands;
       "Unit1.Em6.HmiInterface".cmStackTableGapPadUpDown.commands := "ManualOperationControl_U1Em6".twoWayActuator[6].commands;
   END_REGION
END_REGION

REGION Network 15: Equipment Module 6
   RUNG wire#powerrail
      "CallManualOperationLines_EM"(disableUnit := #disableUnit1, manualOperationEm := "ManualOperationControl_U1Em6".manualOperationEm, manualOperationEmArea := "ManualOperationControl_U1Em6".manualOperationEmArea, manualOperationCms := "ManualOperationControl_U1Em6".manualOperationCms, Axis := "ManualOperationControl_U1Em6".axis, Axis64Pos := "ManualOperationControl_U1Em6".axis64Pos, AxisSfotCam := "ManualOperationControl_U1Em6".softCam, twoWayAcutor := "ManualOperationControl_U1Em6".twoWayActuator, Status := #StatusEm[6].Status, errorID := #errorIDEm[6].errorID)
   END_RUNG
   // the same network as SCL:
   "CallManualOperationLines_EM"(disableUnit := #disableUnit1,
                           manualOperationEm := "ManualOperationControl_U1Em6".manualOperationEm,
                           manualOperationEmArea := "ManualOperationControl_U1Em6".manualOperationEmArea,
                           manualOperationCms := "ManualOperationControl_U1Em6".manualOperationCms,
                           Axis := "ManualOperationControl_U1Em6".axis,
                           Axis64Pos := "ManualOperationControl_U1Em6".axis64Pos,
                           AxisSfotCam := "ManualOperationControl_U1Em6".softCam,
                           twoWayAcutor := "ManualOperationControl_U1Em6".twoWayActuator,
                           Status := #StatusEm[6].Status,
                           errorID := #errorIDEm[6].errorID);
END_REGION

REGION Network 16 (SCL): Equipment Module 7 Cms Mapping
   REGION Input Mapping
       // Axis
       "ManualOperationControl_U1Em7".axis64Pos[6].monitoring := "Unit1.Em7.HmiInterface".cmSepaClampnCutterAxisX.monitoring;
       "ManualOperationControl_U1Em7".axis64Pos[7].monitoring := "Unit1.Em7.HmiInterface".cmSepaClampnCutterAxisZ.monitoring;
       "ManualOperationControl_U1Em7".axis64Pos[8].monitoring := "Unit1.Em7.HmiInterface".cmSepaGripperAxisX.monitoring;
       "ManualOperationControl_U1Em7".axis64Pos[9].monitoring := "Unit1.Em7.HmiInterface".cmSepaGripperAxisZ.monitoring;
       "ManualOperationControl_U1Em7".axis64Pos[10].monitoring := "Unit1.Em7.HmiInterface".cmSepaGripperAxisC.monitoring;
       "ManualOperationControl_U1Em7".axis64Pos[11].monitoring := "Unit1.Em7.HmiInterface".cmJRWinderFrontAxisY.monitoring;
       "ManualOperationControl_U1Em7".axis64Pos[12].monitoring := "Unit1.Em7.HmiInterface".cmJRWinderRearAxisY.monitoring;
       "ManualOperationControl_U1Em7".axis64Pos[13].monitoring := "Unit1.Em7.HmiInterface".cmJRWinderAxisB.monitoring;
       "ManualOperationControl_U1Em7".axis64Pos[14].monitoring := "Unit1.Em7.HmiInterface".cmJRPusherAxisZ.monitoring;

       "ManualOperationControl_U1Em7".axis64Pos[6].configuration := "Unit1.Em7.HmiInterface".cmSepaClampnCutterAxisX.configuration;
       "ManualOperationControl_U1Em7".axis64Pos[7].configuration := "Unit1.Em7.HmiInterface".cmSepaClampnCutterAxisZ.configuration;
       "ManualOperationControl_U1Em7".axis64Pos[8].configuration := "Unit1.Em7.HmiInterface".cmSepaGripperAxisX.configuration;
       "ManualOperationControl_U1Em7".axis64Pos[9].configuration := "Unit1.Em7.HmiInterface".cmSepaGripperAxisZ.configuration;
       "ManualOperationControl_U1Em7".axis64Pos[10].configuration := "Unit1.Em7.HmiInterface".cmSepaGripperAxisC.configuration;
       "ManualOperationControl_U1Em7".axis64Pos[11].configuration := "Unit1.Em7.HmiInterface".cmJRWinderFrontAxisY.configuration;
       "ManualOperationControl_U1Em7".axis64Pos[12].configuration := "Unit1.Em7.HmiInterface".cmJRWinderRearAxisY.configuration;
       "ManualOperationControl_U1Em7".axis64Pos[13].configuration := "Unit1.Em7.HmiInterface".cmJRWinderAxisB.configuration;
       "ManualOperationControl_U1Em7".axis64Pos[14].configuration := "Unit1.Em7.HmiInterface".cmJRPusherAxisZ.configuration;

       // SoftCam
       "ManualOperationControl_U1Em7".softCam[6] := "Unit1.Em7.HmiInterface".cm.softCam.sepaClampnCutterAxisX;
       "ManualOperationControl_U1Em7".softCam[7] := "Unit1.Em7.HmiInterface".cm.softCam.sepaClampnCutterAxisZ;
       "ManualOperationControl_U1Em7".softCam[8] := "Unit1.Em7.HmiInterface".cm.softCam.sepaGripperAxisX;
       "ManualOperationControl_U1Em7".softCam[9] := "Unit1.Em7.HmiInterface".cm.softCam.sepaGripperAxisZ;
       "ManualOperationControl_U1Em7".softCam[10] := "Unit1.Em7.HmiInterface".cm.softCam.sepaGripperAxisC;
       "ManualOperationControl_U1Em7".softCam[11] := "Unit1.Em7.HmiInterface".cm.softCam.jrWinderRearAxisY;
       "ManualOperationControl_U1Em7".softCam[12] := "Unit1.Em7.HmiInterface".cm.softCam.jrWinderFrontAxisY;
       "ManualOperationControl_U1Em7".softCam[13] := "Unit1.Em7.HmiInterface".cm.softCam.jrWinderAxisB;
       "ManualOperationControl_U1Em7".softCam[14] := "Unit1.Em7.HmiInterface".cm.softCam.jrPusherAxisZ;

       // TwoWayActuator
       "ManualOperationControl_U1Em7".twoWayActuator[1].monitoring := "Unit1.Em7.HmiInterface".cmSepaCutterUpDown.monitoring;
       "ManualOperationControl_U1Em7".twoWayActuator[2].monitoring := "Unit1.Em7.HmiInterface".cmSepaClampTopUpDown.monitoring;
       "ManualOperationControl_U1Em7".twoWayActuator[3].monitoring := "Unit1.Em7.HmiInterface".cmSepaClampBottomUpDown.monitoring;
       "ManualOperationControl_U1Em7".twoWayActuator[4].monitoring := "Unit1.Em7.HmiInterface".cmStackGripperOpenClose.monitoring;
       "ManualOperationControl_U1Em7".twoWayActuator[5].monitoring := "Unit1.Em7.HmiInterface".cmStackGripperFwdBwd.monitoring;
       "ManualOperationControl_U1Em7".twoWayActuator[6].monitoring := "Unit1.Em7.HmiInterface".cmJRWinderClampTopRearUpDown.monitoring;
       "ManualOperationControl_U1Em7".twoWayActuator[7].monitoring := "Unit1.Em7.HmiInterface".cmJRWinderClampBtmRearUpDown.monitoring;
       "ManualOperationControl_U1Em7".twoWayActuator[8].monitoring := "Unit1.Em7.HmiInterface".cmJRWinderClampTopFrontUpDown.monitoring;
       "ManualOperationControl_U1Em7".twoWayActuator[9].monitoring := "Unit1.Em7.HmiInterface".cmJRWinderClampBtmFrontUpDown.monitoring;
       "ManualOperationControl_U1Em7".twoWayActuator[10].monitoring := "Unit1.Em7.HmiInterface".cmPusherRollerFwdBwd.monitoring;

   END_REGION


   REGION Output Mapping
       // Axis
       "CallManualOperationLines_ServoPos64Commands"(ManualOperationControl := "ManualOperationControl_U1Em7".axis64Pos[6].commands,
                                                     HmiInterface => "Unit1.Em7.HmiInterface".cmSepaClampnCutterAxisX.commands);

       "CallManualOperationLines_ServoPos64Commands"(ManualOperationControl := "ManualOperationControl_U1Em7".axis64Pos[7].commands,
                                                     HmiInterface => "Unit1.Em7.HmiInterface".cmSepaClampnCutterAxisZ.commands);

       "CallManualOperationLines_ServoPos64Commands"(ManualOperationControl := "ManualOperationControl_U1Em7".axis64Pos[8].commands,
                                                     HmiInterface => "Unit1.Em7.HmiInterface".cmSepaGripperAxisX.commands);

       "CallManualOperationLines_ServoPos64Commands"(ManualOperationControl := "ManualOperationControl_U1Em7".axis64Pos[9].commands,
                                                     HmiInterface => "Unit1.Em7.HmiInterface".cmSepaGripperAxisZ.commands);

       "CallManualOperationLines_ServoPos64Commands"(ManualOperationControl := "ManualOperationControl_U1Em7".axis64Pos[10].commands,
                                                     HmiInterface => "Unit1.Em7.HmiInterface".cmSepaGripperAxisC.commands);

       "CallManualOperationLines_ServoPos64Commands"(ManualOperationControl := "ManualOperationControl_U1Em7".axis64Pos[11].commands,
                                                     HmiInterface => "Unit1.Em7.HmiInterface".cmJRWinderFrontAxisY.commands);

       "CallManualOperationLines_ServoPos64Commands"(ManualOperationControl := "ManualOperationControl_U1Em7".axis64Pos[12].commands,
                                                     HmiInterface => "Unit1.Em7.HmiInterface".cmJRWinderRearAxisY.commands);

       "CallManualOperationLines_ServoPos64Commands"(ManualOperationControl := "ManualOperationControl_U1Em7".axis64Pos[13].commands,
                                                     HmiInterface => "Unit1.Em7.HmiInterface".cmJRWinderAxisB.commands);

       "CallManualOperationLines_ServoPos64Commands"(ManualOperationControl := "ManualOperationControl_U1Em7".axis64Pos[14].commands,
                                                     HmiInterface => "Unit1.Em7.HmiInterface".cmJRPusherAxisZ.commands);

       // TwoWayActuator
       "Unit1.Em7.HmiInterface".cmSepaCutterUpDown.commands := "ManualOperationControl_U1Em7".twoWayActuator[1].commands;
       "Unit1.Em7.HmiInterface".cmSepaClampTopUpDown.commands := "ManualOperationControl_U1Em7".twoWayActuator[2].commands;
       "Unit1.Em7.HmiInterface".cmSepaClampBottomUpDown.commands := "ManualOperationControl_U1Em7".twoWayActuator[3].commands;
       "Unit1.Em7.HmiInterface".cmStackGripperOpenClose.commands := "ManualOperationControl_U1Em7".twoWayActuator[4].commands;
       "Unit1.Em7.HmiInterface".cmStackGripperFwdBwd.commands := "ManualOperationControl_U1Em7".twoWayActuator[5].commands;
       "Unit1.Em7.HmiInterface".cmJRWinderClampTopRearUpDown.commands := "ManualOperationControl_U1Em7".twoWayActuator[6].commands;
       "Unit1.Em7.HmiInterface".cmJRWinderClampBtmRearUpDown.commands := "ManualOperationControl_U1Em7".twoWayActuator[7].commands;
       "Unit1.Em7.HmiInterface".cmJRWinderClampTopFrontUpDown.commands := "ManualOperationControl_U1Em7".twoWayActuator[8].commands;
       "Unit1.Em7.HmiInterface".cmJRWinderClampBtmFrontUpDown.commands := "ManualOperationControl_U1Em7".twoWayActuator[9].commands;
       "Unit1.Em7.HmiInterface".cmPusherRollerFwdBwd.commands := "ManualOperationControl_U1Em7".twoWayActuator[10].commands;

   END_REGION
END_REGION

REGION Network 17: Equipment Module 7
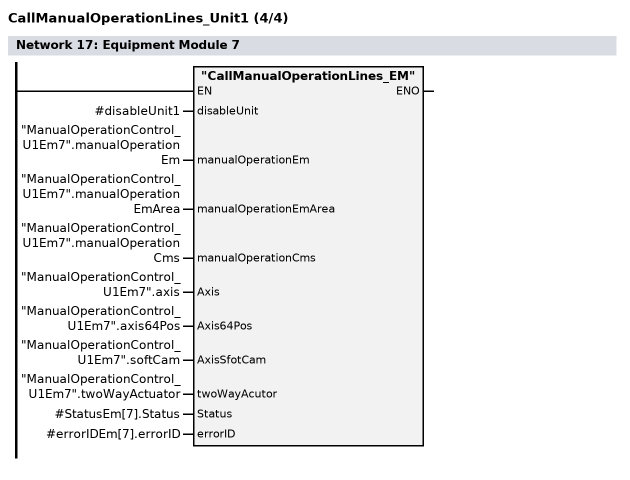
   RUNG wire#powerrail
      "CallManualOperationLines_EM"(disableUnit := #disableUnit1, manualOperationEm := "ManualOperationControl_U1Em7".manualOperationEm, manualOperationEmArea := "ManualOperationControl_U1Em7".manualOperationEmArea, manualOperationCms := "ManualOperationControl_U1Em7".manualOperationCms, Axis := "ManualOperationControl_U1Em7".axis, Axis64Pos := "ManualOperationControl_U1Em7".axis64Pos, AxisSfotCam := "ManualOperationControl_U1Em7".softCam, twoWayAcutor := "ManualOperationControl_U1Em7".twoWayActuator, Status := #StatusEm[7].Status, errorID := #errorIDEm[7].errorID)
   END_RUNG
   // the same network as SCL:
   "CallManualOperationLines_EM"(disableUnit := #disableUnit1,
                           manualOperationEm := "ManualOperationControl_U1Em7".manualOperationEm,
                           manualOperationEmArea := "ManualOperationControl_U1Em7".manualOperationEmArea,
                           manualOperationCms := "ManualOperationControl_U1Em7".manualOperationCms,
                           Axis := "ManualOperationControl_U1Em7".axis,
                           Axis64Pos := "ManualOperationControl_U1Em7".axis64Pos,
                           AxisSfotCam := "ManualOperationControl_U1Em7".softCam,
                           twoWayAcutor := "ManualOperationControl_U1Em7".twoWayActuator,
                           Status := #StatusEm[7].Status,
                           errorID := #errorIDEm[7].errorID);
END_REGION
END_FUNCTION
